{attribute 'qualified_only'}
{attribute 'strict'}
TYPE FSM_States :
(
	Startup_Idle 				:= 1,
	Startup_Power_Check 		:= 2,
	Startup_Breaker_Engage 		:= 3,
	Startup_Control_Power_On 	:= 4,
	Startup_Complete 			:= 5,
	Shutdown_Request 			:= 6,
	Fault_Present 				:= 8,
	Emergency_Stop 				:= 9
);
END_TYPE

(* stored: Version 1.1.0.1, ProductVersion 3.1.4024.15
   DUT FSM_States: Id {c3278140-911d-44c0-b293-1d1a57a5572e} *)
